// TIA Portal project "linia_do_napojow_V18" (V18)

(* hardware
DEVICE "S71500/ET200MP station_1"  S7-1500 station
   slot 0: "Rail_0"  Rack  6ES7 590-1***0-0AA0
   slot 1: "PLC_1"  CPU 1516-3 PN/DP  6ES7 516-3AN02-0AB0  V2.8
      slot 3: "CPU display_1"  6ES7591-1BA00-0AA0
      slot 32768: "PROFINET interface_1"  X1
         slot 32769: "Port_1"  X1 P1
         slot 32770: "Port_2"  X1 P2
      slot 33024: "PROFINET interface_2"  X2
         slot 33025: "Port_1"  X2 P1
      slot 33280: "DP interface_1"  X3
      slot 34817: "Virtual CP interface port_1"  Virtual CP interface port  Virtual CP interface port
   slot 2: "DI 32x24VDC HF_1"  DI 32x24VDC HF  6ES7 521-1BL00-0AB0  V2.2
   slot 3: "DQ 32x24VDC/0.5A HF_1"  DQ 32x24VDC/0.5A HF  6ES7 522-1BL01-0AB0  V1.1
   slot 4: "AI 8xU/I/RTD/TC ST_1"  AI 8xU/I/RTD/TC ST  6ES7 531-7KF00-0AB0  V2.2
   slot 5: "AQ 4xU/I ST_1"  AQ 4xU/I ST  6ES7 532-5HD00-0AB0  V2.2
DEVICE "HMI_1"  KTP900 Basic PN
   slot 0: "HMI_1"  KTP900 Basic PN  6AV2 123-2JB03-0AX0  16.0.0.0
   slot 1: "HMI_RT_1"  KTP900 Basic PN  6AV2 123-2JB03-0AX0  16.0.0.0
   slot 5: "HMI_1.IE_CP_1"  PROFINET Interface  16.0.0.0
      slot 1: "PROFINET Interface_1"  PROFINET Interface
         slot 1: "Port_1"  Port
*)

// ===== PLC "PLC_1"  CPU 1516-3 PN/DP =====

VAR_GLOBAL   // PLC tag table "Default tag table"
   "System_Byte" AT %MB1 : Byte;
   "FirstScan" AT %M1.0 : Bool;
   "DiagStatusUpdate" AT %M1.1 : Bool;
   "AlwaysTRUE" AT %M1.2 : Bool;
   "AlwaysFALSE" AT %M1.3 : Bool;
   "Clock_Byte" AT %MB0 : Byte;
   "Clock_10Hz" AT %M0.0 : Bool;
   "Clock_5Hz" AT %M0.1 : Bool;
   "Clock_2.5Hz" AT %M0.2 : Bool;
   "Clock_2Hz" AT %M0.3 : Bool;
   "Clock_1.25Hz" AT %M0.4 : Bool;
   "Clock_1Hz" AT %M0.5 : Bool;
   "Clock_0.625Hz" AT %M0.6 : Bool;
   "Clock_0.5Hz" AT %M0.7 : Bool;
   "rozlaczenie_tasmy" AT %M100.2 : Bool;
   "reset_licznika" AT %M100.3 : Bool;
   "zatrzymanie_tasmy" AT %M101.2 : Bool;
   "ilosc_butelek" AT %MW10 : Int;
   "reset_licznika_zak" AT %M101.3 : Bool;
   "ilosc_butelek_zak" AT %MW16 : Int;
   "Wylacznik_bezpieczenstwa" AT %M205.0 : Bool;
   "Wlacznik/Wylacznik_glowny" AT %M206.0 : Bool;
   "start_przenosik" AT %M204.0 : Bool;
   "stop_przenosnik" AT %M204.1 : Bool;
   "przenosnik_tasmowy" AT %Q1.4 : Bool;
   "wylacznik_przenosnika_tasmowego" AT %I1.4 : Bool;
   "wylacznik_nalewarki" AT %I1.5 : Bool;
   "wylacznik_zakrecarki" AT %I1.6 : Bool;
   "wylacznik_etykieciarki" AT %I1.7 : Bool;
   "wylacznik_pakowanie" AT %I2.0 : Bool;
   "samopod_start_zak" AT %M102.3 : Bool;
   "samopod_start_nal" AT %M100.4 : Bool;
   "Wlacznik_500ml" AT %M207.0 : Bool;
   "silownik" AT %Q1.5 : Bool;
   "sygnalizator_dzwiekowy" AT %Q2.2 : Bool;
   "robot" AT %Q2.3 : Bool;
   "lampa_przenosnik" AT %Q2.4 : Bool;
   "licznik_etykiet" AT %MW50 : Int;
   "cz_poj_ety" AT %M210.0 : Bool;
   "reset_licznika_etyk" AT %M211.0 : Bool;
   "pamiec_smakow" AT %M100.5 : Bool;
   "smak_zatrzymaj" AT %M212.2 : Bool;
   "czas_nalewarka" AT %MD300 : Time;
   "czas_pakowanie" AT %MD304 : Time;
   "czas_zakrecarka" AT %MD308 : Time;
   "cz_butelek_pakowanie" AT %M230.0 : Bool;
   "Tag_1" AT %MW400 : Word;
   "licznik_przenosnik" AT %MW30 : Int;
   "res_licz_przen" AT %M350.0 : Bool;
   "Tag_4" AT %MD32 : Time;
   "Tag_5" AT %M500.0 : Bool;
   "res_licz_nalew" AT %M350.1 : Bool;
   "licznik_nalewarak" AT %MW34 : Int;
   "Tag_2" AT %M350.2 : Bool;
   "Tag_3" AT %MW38 : Word;
   "czas_move" AT %MD312 : DWord;
   "czas_w_int" AT %MD316 : UDInt;
   "Tag_6" AT %M320.0 : Bool;
   "Tag_7" AT %MD321 : Time;
   "Tag_8" AT %MD325 : Time;
   "Tag_9" AT %MD329 : DInt;
   "Tag_10" AT %I90.0 : Bool;
END_VAR

VAR_GLOBAL   // PLC tag table "Nalewarka"
   "start_nalewarka" AT %M100.0 : Bool;
   "stop_nalewarka" AT %M100.1 : Bool;
   "cz_pojemnosciowy" AT %M200.0 : Bool;
   "dozy" AT %Q0.1 : Bool;
   "tasma" AT %Q0.0 : Bool;
   "lampa" AT %Q0.2 : Bool;
   "wl_pomarancza" AT %M212.0 : Bool;
   "pomarancza" AT %Q2.5 : Bool;
   "wl_truskawka" AT %M212.1 : Bool;
   "truskawka" AT %Q2.6 : Bool;
   "cz_poz_napoju" AT %M213.0 : Bool;
END_VAR

VAR_GLOBAL   // PLC tag table "Zakrecarka"
   "start_zakrecarka" AT %M101.0 : Bool;
   "stop_zakrecarka" AT %M101.1 : Bool;
   "cz_pojemnosciowy_zak" AT %M201.0 : Bool;
   "tasma_zakrecarka" AT %Q0.4 : Bool;
   "zakretka" AT %Q0.3 : Bool;
   "lampa_sygnalizacyjna" AT %Q0.5 : Bool;
END_VAR

VAR_GLOBAL   // PLC tag table "Etykieciarka"
   "start_etykieciarka" AT %M102.0 : Bool;
   "stop_etykieciarka" AT %M102.1 : Bool;
   "cz_swiatlowodowy" AT %M202.0 : Bool;
   "etykieta" AT %Q0.6 : Bool;
   "tasma_etykieciarka" AT %Q0.7 : Bool;
   "lampa_sygnalizacyjna_etyk" AT %Q1.0 : Bool;
END_VAR

VAR_GLOBAL   // PLC tag table "Pakowanie"
   "start_pakowaie" AT %M103.0 : Bool;
   "stop_pakowanie" AT %M103.1 : Bool;
   "cz_pojemnosciowy_pak" AT %M203.0 : Bool;
   "tasma_pakowanie" AT %Q1.2 : Bool;
   "lampa_sygnalizacyjna_pak" AT %Q1.1 : Bool;
   "cz_do_robota" AT %Q1.3 : Bool;
END_VAR

DATA_BLOCK "Nalewarka_DB"   // DB3
{ S7_Optimized_Access := 'TRUE' }
VERSION : 0.1
// stored: InstanceOfName Nalewarka
"Nalewarka"
BEGIN
END_DATA_BLOCK

DATA_BLOCK "Zakrecarka_DB"   // DB6
{ S7_Optimized_Access := 'TRUE' }
VERSION : 0.1
// stored: InstanceOfName Zakrecarka
"Zakrecarka"
BEGIN
END_DATA_BLOCK

DATA_BLOCK "Etykieciarka_DB"   // DB7
{ S7_Optimized_Access := 'TRUE' }
VERSION : 0.1
// stored: InstanceOfName Etykieciarka
"Etykieciarka"
BEGIN
END_DATA_BLOCK

DATA_BLOCK "Pakowanie_DB"   // DB9
{ S7_Optimized_Access := 'TRUE' }
VERSION : 0.1
// stored: InstanceOfName Pakowanie
"Pakowanie"
BEGIN
END_DATA_BLOCK

DATA_BLOCK "Przenosnik tasmowy_DB"   // DB12
{ S7_Optimized_Access := 'TRUE' }
VERSION : 0.1
// stored: InstanceOfName Przenosnik tasmowy
"Przenosnik tasmowy"
BEGIN
END_DATA_BLOCK

// folder: System blocks/Program resources

DATA_BLOCK "IEC_Counter_0_DB"   // DB1
{ S7_Optimized_Access := 'TRUE' }
AUTHOR : Simatic
FAMILY : IEC
NAME : CNTR
VERSION : 1.0
// stored: InstanceOfName IEC_COUNTER
"IEC_COUNTER"
BEGIN
END_DATA_BLOCK

DATA_BLOCK "IEC_Timer_0_DB"   // DB2
{ S7_Optimized_Access := 'TRUE' }
AUTHOR : Simatic
FAMILY : IEC
NAME : IEC_TMR
VERSION : 1.0
// stored: InstanceOfName IEC_TIMER
"IEC_TIMER"
BEGIN
END_DATA_BLOCK

DATA_BLOCK "IEC_Counter_0_DB_1"   // DB4
{ S7_Optimized_Access := 'TRUE' }
AUTHOR : Simatic
FAMILY : IEC
NAME : CNTR
VERSION : 1.0
// stored: InstanceOfName IEC_COUNTER
"IEC_COUNTER"
BEGIN
END_DATA_BLOCK

DATA_BLOCK "IEC_Timer_0_DB_1"   // DB5
{ S7_Optimized_Access := 'TRUE' }
AUTHOR : Simatic
FAMILY : IEC
NAME : IEC_TMR
VERSION : 1.0
// stored: InstanceOfName IEC_TIMER
"IEC_TIMER"
BEGIN
END_DATA_BLOCK

DATA_BLOCK "IEC_Counter_0_DB_2"   // DB8
{ S7_Optimized_Access := 'TRUE' }
AUTHOR : Simatic
FAMILY : IEC
NAME : CNTR
VERSION : 1.0
// stored: InstanceOfName IEC_COUNTER
"IEC_COUNTER"
BEGIN
END_DATA_BLOCK

DATA_BLOCK "IEC_Timer_0_DB_2"   // DB10
{ S7_Optimized_Access := 'TRUE' }
AUTHOR : Simatic
FAMILY : IEC
NAME : IEC_TMR
VERSION : 1.0
// stored: InstanceOfName IEC_TIMER
"IEC_TIMER"
BEGIN
END_DATA_BLOCK

// folder: (top level)

FUNCTION_BLOCK "Nalewarka"   // FB1, LAD
{ S7_Optimized_Access := 'TRUE' }
VERSION : 0.1
   VAR
      czas_nalewarka : Time;
   END_VAR
   VAR_TEMP   // added for the SCL form of the ladder/FBD networks
      _w1 : Bool;
   END_VAR
BEGIN

REGION Network 1
   // Start przenośnika taśmowego i zapalenie się lampy sygnalizacyjnej.
   // Wyłącznik nalewarki znajduje się fizycznie na linii produkcyjnej, w jego skład wchodzi również system ryglowania. Stop natomiast w panelu HMI.
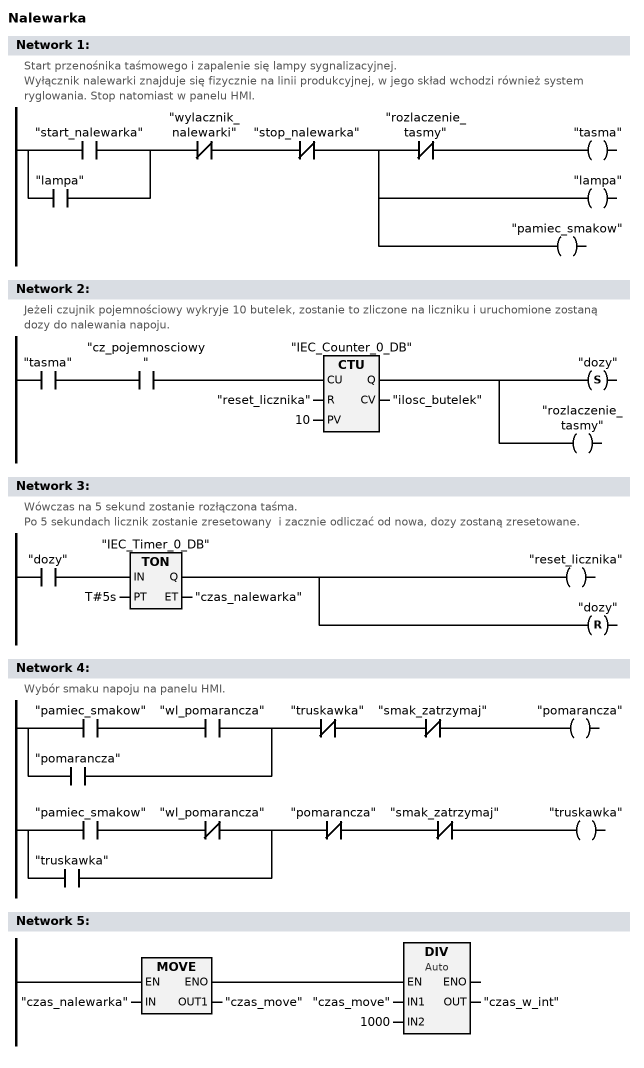
   RUNG wire#powerrail
      Contact( "start_nalewarka" )
      wire#w1
      I_Contact( "wylacznik_nalewarki" )
      I_Contact( "stop_nalewarka" )
      wire#w2
      I_Contact( "rozlaczenie_tasmy" )
      Coil( "tasma" )
   END_RUNG
   RUNG wire#powerrail
      Contact( "lampa" )
   END_RUNG wire#w1
   RUNG wire#w2
      Coil( "lampa" )
   END_RUNG
   RUNG wire#w2
      Coil( "pamiec_smakow" )
   END_RUNG
   // the same network as SCL:
   #_w1 := ("start_nalewarka" OR "lampa") AND NOT "wylacznik_nalewarki" AND NOT "stop_nalewarka";
   "tasma" := #_w1 AND NOT "rozlaczenie_tasmy";
   "lampa" := #_w1;
   "pamiec_smakow" := #_w1;
END_REGION

REGION Network 2
   // Jeżeli czujnik pojemnościowy wykryje 10 butelek, zostanie to zliczone na liczniku i uruchomione zostaną dozy do nalewania napoju.
   "IEC_Counter_0_DB".CTU(CU := "tasma" AND "cz_pojemnosciowy",
                          R := "reset_licznika",
                          PV := 10,
                          CV => "ilosc_butelek");
   IF "IEC_Counter_0_DB".Q THEN "dozy" := TRUE; END_IF;
   "rozlaczenie_tasmy" := "IEC_Counter_0_DB".Q;
END_REGION

REGION Network 3
   // Wówczas na 5 sekund zostanie rozłączona taśma.
   // Po 5 sekundach licznik zostanie zresetowany  i zacznie odliczać od nowa, dozy zostaną zresetowane.
   "IEC_Timer_0_DB".TON(IN := "dozy", PT := T#5s, ET => "czas_nalewarka");
   "reset_licznika" := "IEC_Timer_0_DB".Q;
   IF "IEC_Timer_0_DB".Q THEN "dozy" := FALSE; END_IF;
END_REGION

REGION Network 4
   // Wybór smaku napoju na panelu HMI.
   RUNG wire#powerrail
      Contact( "pamiec_smakow" )
      Contact( "wl_pomarancza" )
      wire#w1
      I_Contact( "truskawka" )
      I_Contact( "smak_zatrzymaj" )
      Coil( "pomarancza" )
   END_RUNG
   RUNG wire#powerrail
      Contact( "pomarancza" )
   END_RUNG wire#w1
   RUNG wire#powerrail
      Contact( "pamiec_smakow" )
      I_Contact( "wl_pomarancza" )
      wire#w2
      I_Contact( "pomarancza" )
      I_Contact( "smak_zatrzymaj" )
      Coil( "truskawka" )
   END_RUNG
   RUNG wire#powerrail
      Contact( "truskawka" )
   END_RUNG wire#w2
   // the same network as SCL:
   "pomarancza" := (("pamiec_smakow" AND "wl_pomarancza") OR "pomarancza") AND NOT "truskawka" AND NOT "smak_zatrzymaj";
   "truskawka" := (("pamiec_smakow" AND NOT "wl_pomarancza") OR "truskawka") AND NOT "pomarancza" AND NOT "smak_zatrzymaj";
END_REGION

REGION Network 5
   RUNG wire#powerrail
      Move(in := "czas_nalewarka", out1 => "czas_move")
      Div(in1 := "czas_move", in2 := 1000, out => "czas_w_int")
   END_RUNG
   // the same network as SCL:
   "czas_move" := "czas_nalewarka";
   "czas_w_int" := "czas_move" / 1000;
END_REGION
END_FUNCTION_BLOCK

FUNCTION_BLOCK "Zakrecarka"   // FB2, LAD
{ S7_Optimized_Access := 'TRUE' }
VERSION : 0.1
   VAR_TEMP   // added for the SCL form of the ladder/FBD networks
      _w1 : Bool;
   END_VAR
BEGIN

REGION Network 1
   // Start przenośnika taśmowego i zapalenie się lampy sygnalizacyjnej.
   // Wyłącznik zakręcarki znajduje się fizycznie na linii produkcyjnej, w jego skład wchodzi również system ryglowania. Stop natomiast w panelu HMI.
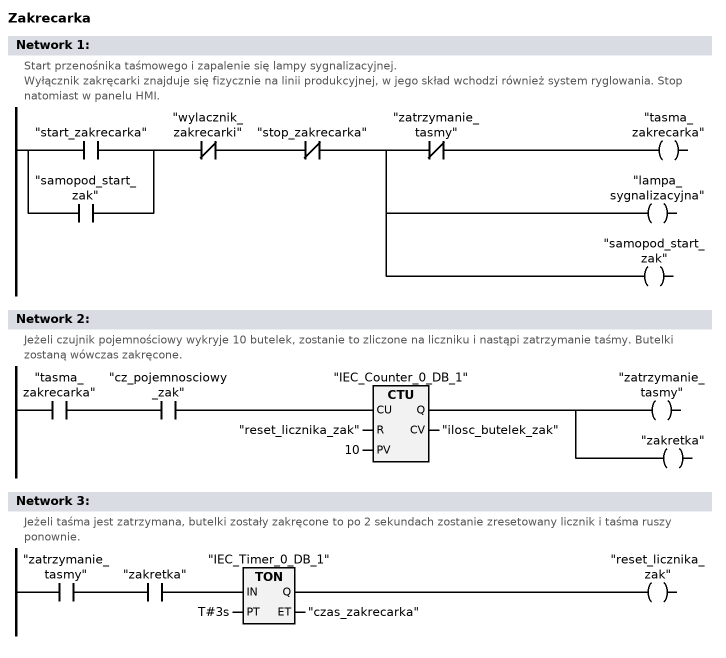
   RUNG wire#powerrail
      Contact( "start_zakrecarka" )
      wire#w1
      I_Contact( "wylacznik_zakrecarki" )
      I_Contact( "stop_zakrecarka" )
      wire#w2
      I_Contact( "zatrzymanie_tasmy" )
      Coil( "tasma_zakrecarka" )
   END_RUNG
   RUNG wire#powerrail
      Contact( "samopod_start_zak" )
   END_RUNG wire#w1
   RUNG wire#w2
      Coil( "lampa_sygnalizacyjna" )
   END_RUNG
   RUNG wire#w2
      Coil( "samopod_start_zak" )
   END_RUNG
   // the same network as SCL:
   #_w1 := ("start_zakrecarka" OR "samopod_start_zak") AND NOT "wylacznik_zakrecarki" AND NOT "stop_zakrecarka";
   "tasma_zakrecarka" := #_w1 AND NOT "zatrzymanie_tasmy";
   "lampa_sygnalizacyjna" := #_w1;
   "samopod_start_zak" := #_w1;
END_REGION

REGION Network 2
   // Jeżeli czujnik pojemnościowy wykryje 10 butelek, zostanie to zliczone na liczniku i nastąpi zatrzymanie taśmy. Butelki zostaną wówczas zakręcone.
   "IEC_Counter_0_DB_1".CTU(CU := "tasma_zakrecarka" AND "cz_pojemnosciowy_zak",
                           R := "reset_licznika_zak",
                           PV := 10,
                           CV => "ilosc_butelek_zak");
   "zatrzymanie_tasmy" := "IEC_Counter_0_DB_1".Q;
   "zakretka" := "IEC_Counter_0_DB_1".Q;
END_REGION

REGION Network 3
   // Jeżeli taśma jest zatrzymana, butelki zostały zakręcone to po 2 sekundach zostanie zresetowany licznik i taśma ruszy ponownie.
   "IEC_Timer_0_DB_1".TON(IN := "zatrzymanie_tasmy" AND "zakretka", PT := T#3s, ET => "czas_zakrecarka");
   "reset_licznika_zak" := "IEC_Timer_0_DB_1".Q;
END_REGION
END_FUNCTION_BLOCK

FUNCTION_BLOCK "Etykieciarka"   // FB3, LAD
{ S7_Optimized_Access := 'TRUE' }
VERSION : 0.1
BEGIN

REGION Network 1
   // Start przenośnika taśmowego i zapalenie się lampy sygnalizacyjnej.
   // Wyłącznik etykieciarki znajduje się fizycznie na linii produkcyjnej. Stop natomiast w panelu HMI.
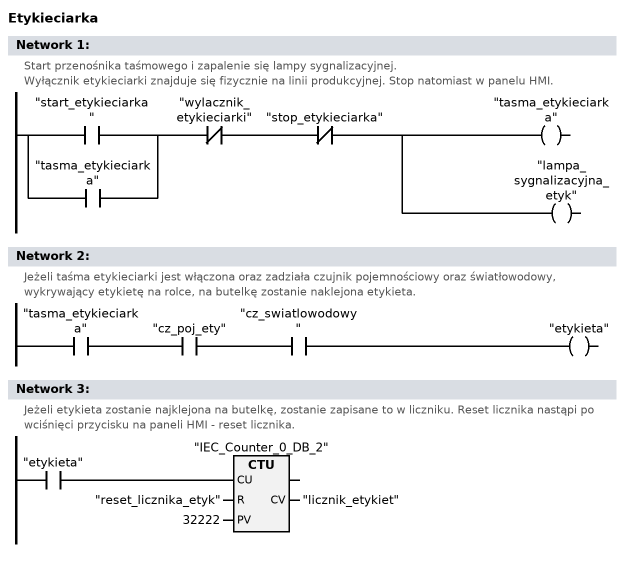
   RUNG wire#powerrail
      Contact( "start_etykieciarka" )
      wire#w1
      I_Contact( "wylacznik_etykieciarki" )
      I_Contact( "stop_etykieciarka" )
      wire#w2
      Coil( "tasma_etykieciarka" )
   END_RUNG
   RUNG wire#powerrail
      Contact( "tasma_etykieciarka" )
   END_RUNG wire#w1
   RUNG wire#w2
      Coil( "lampa_sygnalizacyjna_etyk" )
   END_RUNG
   // the same network as SCL:
   "tasma_etykieciarka" := ("start_etykieciarka" OR "tasma_etykieciarka") AND NOT "wylacznik_etykieciarki" AND NOT "stop_etykieciarka";
   "lampa_sygnalizacyjna_etyk" := "tasma_etykieciarka";
END_REGION

REGION Network 2
   // Jeżeli taśma etykieciarki jest włączona oraz zadziała czujnik pojemnościowy oraz światłowodowy, wykrywający etykietę na rolce, na butelkę zostanie naklejona etykieta.
   RUNG wire#powerrail
      Contact( "tasma_etykieciarka" )
      Contact( "cz_poj_ety" )
      Contact( "cz_swiatlowodowy" )
      Coil( "etykieta" )
   END_RUNG
   // the same network as SCL:
   "etykieta" := "tasma_etykieciarka" AND "cz_poj_ety" AND "cz_swiatlowodowy";
END_REGION

REGION Network 3
   // Jeżeli etykieta zostanie najklejona na butelkę, zostanie zapisane to w liczniku. Reset licznika nastąpi po wciśnięci przycisku na paneli HMI - reset licznika.
   "IEC_Counter_0_DB_2".CTU(CU := "etykieta", R := "reset_licznika_etyk", PV := 32222, CV => "licznik_etykiet");
END_REGION
END_FUNCTION_BLOCK

FUNCTION_BLOCK "Pakowanie"   // FB4, LAD
{ S7_Optimized_Access := 'TRUE' }
VERSION : 0.1
BEGIN

REGION Network 1
   // Start przenośnika taśmowego i zapalenie się lampy sygnalizacyjnej.
   // Wyłącznik pakowania znajduje się fizycznie na linii produkcyjnej, w jego skład wchodzi również kurtyna świetlna. Stop natomiast w panelu HMI.
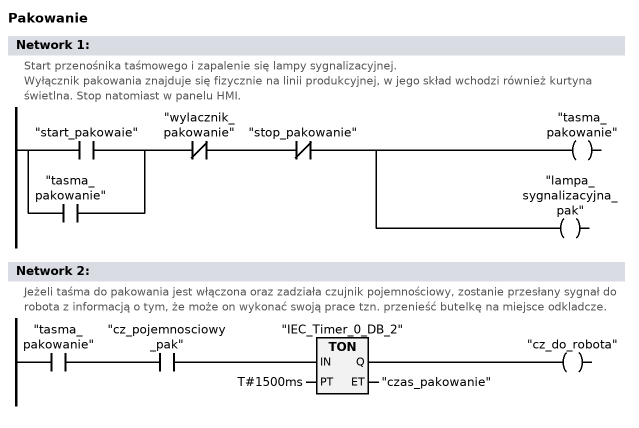
   RUNG wire#powerrail
      Contact( "start_pakowaie" )
      wire#w1
      I_Contact( "wylacznik_pakowanie" )
      I_Contact( "stop_pakowanie" )
      wire#w2
      Coil( "tasma_pakowanie" )
   END_RUNG
   RUNG wire#powerrail
      Contact( "tasma_pakowanie" )
   END_RUNG wire#w1
   RUNG wire#w2
      Coil( "lampa_sygnalizacyjna_pak" )
   END_RUNG
   // the same network as SCL:
   "tasma_pakowanie" := ("start_pakowaie" OR "tasma_pakowanie") AND NOT "wylacznik_pakowanie" AND NOT "stop_pakowanie";
   "lampa_sygnalizacyjna_pak" := "tasma_pakowanie";
END_REGION

REGION Network 2
   // Jeżeli taśma do pakowania jest włączona oraz zadziała czujnik pojemnościowy, zostanie przesłany sygnał do robota z informacją o tym, że może on wykonać swoją prace tzn. przenieść butelkę na miejsce odkladcze.
   "IEC_Timer_0_DB_2".TON(IN := "tasma_pakowanie" AND "cz_pojemnosciowy_pak",
                          PT := T#1500ms,
                          ET => "czas_pakowanie");
   "cz_do_robota" := "IEC_Timer_0_DB_2".Q;
END_REGION
END_FUNCTION_BLOCK

FUNCTION_BLOCK "Przenosnik tasmowy"   // FB5, LAD
{ S7_Optimized_Access := 'TRUE' }
VERSION : 0.1
   VAR_TEMP
      mem0 : Time;
   END_VAR
BEGIN

REGION Network 1
   // Start przenośnika taśmowego.
   // Wyłącznik przenośnika znajduje się fizycznie na linii produkcyjnej. Stop natomiast w panelu HMI.
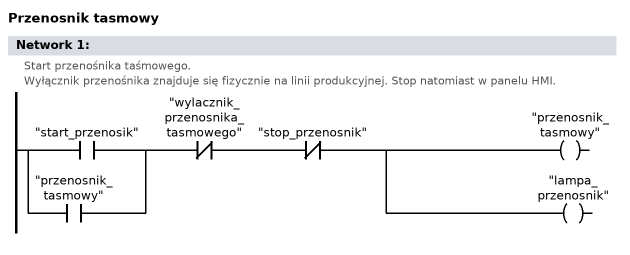
   RUNG wire#powerrail
      Contact( "start_przenosik" )
      wire#w1
      I_Contact( "wylacznik_przenosnika_tasmowego" )
      I_Contact( "stop_przenosnik" )
      wire#w2
      Coil( "przenosnik_tasmowy" )
   END_RUNG
   RUNG wire#powerrail
      Contact( "przenosnik_tasmowy" )
   END_RUNG wire#w1
   RUNG wire#w2
      Coil( "lampa_przenosnik" )
   END_RUNG
   // the same network as SCL:
   "przenosnik_tasmowy" := ("start_przenosik" OR "przenosnik_tasmowy") AND NOT "wylacznik_przenosnika_tasmowego" AND NOT "stop_przenosnik";
   "lampa_przenosnik" := "przenosnik_tasmowy";
END_REGION
END_FUNCTION_BLOCK

ORGANIZATION_BLOCK "Main"   // OB1, LAD, ProgramCycle
TITLE = "Main Program Sweep (Cycle)"
{ S7_Optimized_Access := 'TRUE' }
VERSION : 0.1
   VAR_INPUT
      Initial_Call : Bool;   // Initial call of this OB
      Remanence : Bool;   // =True, if remanent data are available
   END_VAR
   VAR_TEMP   // added for the SCL form of the ladder/FBD networks
      _w1 : Bool;
      _w2 : Bool;
      _w3 : Bool;
      _w4 : Bool;
      _w5 : Bool;
   END_VAR
BEGIN

REGION Network 1
   // Linię produkcyjną uruchamiamy poprzez włącznik główny oraz dodatkowo każdy etap produkcji na panelu HMI.
   // Wyłącznik bezpieczeństwa znajduje się w kilku miejscach na linii produkcyjnej.
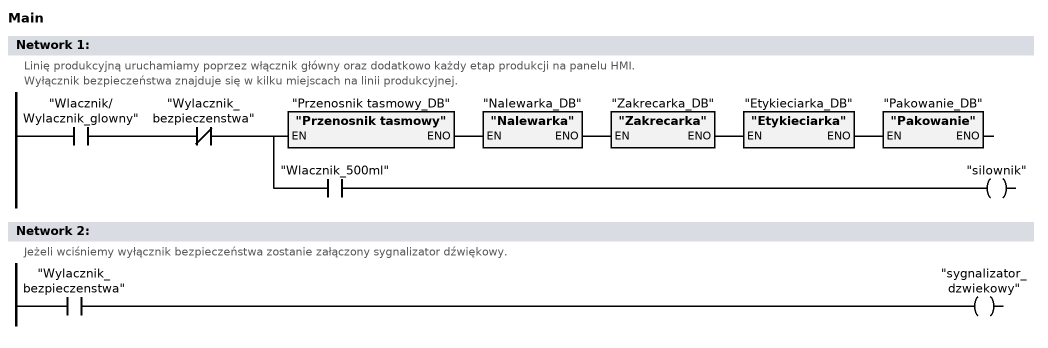
   RUNG wire#powerrail
      Contact( "Wlacznik/Wylacznik_glowny" )
      I_Contact( "Wylacznik_bezpieczenstwa" )
      wire#w1
      "Przenosnik tasmowy_DB"()
      "Nalewarka_DB"()
      "Zakrecarka_DB"()
      "Etykieciarka_DB"()
      "Pakowanie_DB"()
   END_RUNG
   RUNG wire#w1
      Contact( "Wlacznik_500ml" )
      Coil( "silownik" )
   END_RUNG
   // the same network as SCL:
   #_w1 := "Wlacznik/Wylacznik_glowny" AND NOT "Wylacznik_bezpieczenstwa";
   "Przenosnik tasmowy_DB"(EN := #_w1, ENO => #_w2);   // "Przenosnik tasmowy"
   "Nalewarka_DB"(EN := #_w2, ENO => #_w3);   // "Nalewarka"
   "Zakrecarka_DB"(EN := #_w3, ENO => #_w4);   // "Zakrecarka"
   "Etykieciarka_DB"(EN := #_w4, ENO => #_w5);   // "Etykieciarka"
   IF #_w5 THEN
       "Pakowanie_DB"();   // "Pakowanie"
   END_IF;
   "silownik" := #_w1 AND "Wlacznik_500ml";
END_REGION

REGION Network 2
   // Jeżeli wciśniemy wyłącznik bezpieczeństwa zostanie załączony sygnalizator dźwiękowy.
   RUNG wire#powerrail
      Contact( "Wylacznik_bezpieczenstwa" )
      Coil( "sygnalizator_dzwiekowy" )
   END_RUNG
   // the same network as SCL:
   "sygnalizator_dzwiekowy" := "Wylacznik_bezpieczenstwa";
END_REGION
END_ORGANIZATION_BLOCK

(* ===== HMI "HMI_RT_1" =====
system functions are stored by id; their names below are inferred from use
connection "HMI_Connection_1": ETHERNET, SMART_S7_1500_OMS

HMI tags "Default tag table"
   "Wlacznik_glowny" : Bool = PLC "Wlacznik/Wylacznik_glowny" AT %M206.0, 1 s
   "start_przenosik" : Bool = PLC start_przenosik AT %M204.0, 1 s
   "stop_przenosnik" : Bool = PLC stop_przenosnik AT %M204.1, 1 s
   "przenosnik_tasmowy" : Bool = PLC przenosnik_tasmowy AT %Q1.4, 1 s
      on ChangeValue: function_b9b71300("MOVE(1)", 1)
   "start_nalewarka" : Bool = PLC start_nalewarka AT %M100.0, 1 s
   "stop_nalewarka" : Bool = PLC stop_nalewarka AT %M100.1, 1 s
   "start_zakrecarka" : Bool = PLC start_zakrecarka AT %M101.0, 1 s
   "stop_zakrecarka" : Bool = PLC stop_zakrecarka AT %M101.1, 1 s
   "start_etykieciarka" : Bool = PLC start_etykieciarka AT %M102.0, 1 s
   "stop_etykieciarka" : Bool = PLC stop_etykieciarka AT %M102.1, 1 s
   "start_pakowaie" : Bool = PLC start_pakowaie AT %M103.0, 1 s
   "stop_pakowanie" : Bool = PLC stop_pakowanie AT %M103.1, 1 s
   "silownik" : Bool = PLC silownik AT %Q1.5, 1 s
   "Wlacznik_500ml" : Bool = PLC Wlacznik_500ml AT %M207.0, 1 s
   "lampa" : Bool = PLC lampa AT %Q0.2, 1 s
   "lampa_sygnalizacyjna" : Bool = PLC lampa_sygnalizacyjna AT %Q0.5, 1 s
   "lampa_sygnalizacyjna_etyk" : Bool = PLC lampa_sygnalizacyjna_etyk AT %Q1.0, 1 s
   "lampa_sygnalizacyjna_pak" : Bool = PLC lampa_sygnalizacyjna_pak AT %Q1.1, 1 s
   "cz_do_robota" : Bool = PLC cz_do_robota AT %Q1.3, 1 s
   "tasma_pakowanie" : Bool = PLC tasma_pakowanie AT %Q1.2, 1 s
      on ChangeValue: function_b9b71300("move_pako", 1)
   "cz_pojemnosciowy" : Bool = PLC cz_pojemnosciowy AT %M200.0, 1 s
   "dozy" : Bool = PLC dozy AT %Q0.1, 1 s
   "tasma" : Bool = PLC tasma AT %Q0.0, 1 s
      on ChangeValue: function_b9b71300("MOVE_nal", 1)
   "ilosc_butelek" : Int = PLC ilosc_butelek AT %MW10, 1 s
   "cz_pojemnosciowy_pak" : Bool = PLC cz_pojemnosciowy_pak AT %M203.0, 1 s
   "lampa_przenosnik" : Bool = PLC lampa_przenosnik AT %Q2.4, 1 s
   "licznik_etykiet" : Int = PLC licznik_etykiet AT %MW50, 1 s
   "tasma_etykieciarka" : Bool = PLC tasma_etykieciarka AT %Q0.7, 1 s
      on ChangeValue: function_b9b71300("move_etyk", 1)
   "cz_poj_ety" : Bool = PLC cz_poj_ety AT %M210.0, 1 s
   "cz_swiatlowodowy" : Bool = PLC cz_swiatlowodowy AT %M202.0, 1 s
   "etykieta" : Bool = PLC etykieta AT %Q0.6, 1 s
   "reset_licznika_etyk" : Bool = PLC reset_licznika_etyk AT %M211.0, 1 s
   "ilosc_butelek_zak" : Int = PLC ilosc_butelek_zak AT %MW16, 1 s
   "tasma_zakrecarka" : Bool = PLC tasma_zakrecarka AT %Q0.4, 1 s
      on ChangeValue: function_b9b71300("move_zak", 1)
   "cz_pojemnosciowy_zak" : Bool = PLC cz_pojemnosciowy_zak AT %M201.0, 1 s
   "zakretka" : Bool = PLC zakretka AT %Q0.3, 1 s
   "wl_pomarancza" : Bool = PLC wl_pomarancza AT %M212.0, 1 s
   "sygnalizator_dzwiekowy" : Bool = PLC sygnalizator_dzwiekowy AT %Q2.2, 1 s
   "smak_zatrzymaj" : Bool = PLC smak_zatrzymaj AT %M212.2, 1 s
   "pomarancza" : Bool = PLC pomarancza AT %Q2.5, 1 s
   "truskawka" : Bool = PLC truskawka AT %Q2.6, 1 s
   "czas_pakowanie" : Time = PLC czas_pakowanie AT %MD304, 1 s
   "czas_zakrecarka" : Time = PLC czas_zakrecarka AT %MD308, 1 s
   "czas_nalewarka" : Time = PLC czas_nalewarka AT %MD300, 1 s
   "move" : Int, internal
   "Clock_Byte" : Byte = PLC Clock_Byte AT %MB0, 1 s
   "Tag_1" : Word = PLC Tag_1 AT %MW400, 1 s
   "Tag_2" : Int = PLC licznik_przenosnik AT %MW30, 1 s
   "Tag_4" : Time = PLC Tag_4 AT %MD32, 1 s
   "licznik_nalewarak" : Int = PLC licznik_nalewarak AT %MW34, 1 s
   "MOVE(1)" : Int, internal
   "MOVE_nal" : Int, internal
   "rozlaczenie_tasmy" : Bool = PLC rozlaczenie_tasmy AT %M100.2, 1 s
   "Tag_6" : DWord = PLC czas_move AT %MD312, 1 s
   "Tag_7" : UDInt = PLC czas_w_int AT %MD316, 1 s
   "move_etyk" : Int, internal
   "Tag_6(1)" : Bool = PLC Tag_6 AT %M320.0, 1 s
   "Tag_7(1)" : Time = PLC Tag_7 AT %MD321, 1 s
   "Tag_9" : DInt = PLC Tag_9 AT %MD329, 1 s
   "move_zak" : Int, internal
   "move_nal(1)" : Int, internal
   "move_pako" : Int, internal

text list "Lista": 0 'Butelki szklane - 250ml'; 1 'Butelki szklane - 500ml'

text list "Smaki": 0 'truskawkowy'; 1 'pomarańczowy'

text list "Ilosc_butelek": 1 '10'; 2 '9'; 3 '8'; 4 '7'; 5 '6'; 6 '5'; 7 '4'; 8 '3'; 9 '2'; 10 '1'

Template "Template_1" 800x480
   Button "Exit" at 722,440 size 55x39; TextOff 'Exit'; PictureOff "ExitRuntime_KTP900_Basic_PN_TR"; PictureOn "ExitRuntime_KTP900_Basic_PN_TR"
      on Release: StopRuntime(0)
   Button "Template_Button" at 622,440 size 55x39; TextOff 'Text'
   Button "Template_Button_1" at 522,440 size 55x39; TextOff 'Text'
   Button "Template_Button_2" at 422,440 size 55x39; TextOff 'Text'
   Button "Template_Button_3" at 322,440 size 55x39; TextOff 'Text'
   Button "Template_Button_4" at 222,440 size 55x39; TextOff 'Text'
   Button "Alarms" at 122,440 size 55x39; TextOff 'Alarms'; PictureOff "AlarmDisplay_KTP900_Basic_PN_TR"; PictureOn "AlarmDisplay_KTP900_Basic_PN_TR"
      on Release: function_ef3f5d25("Alarm window_Unacknowledged", -1)
   Button "Start screen" at 22,440 size 55x39; TextOff 'Start screen'; PictureOff "NavigateHome_KTP900_Basic_PN_TR"; PictureOn "NavigateHome_KTP900_Basic_PN_TR"
      on Release: ActivateScreen("Wyswietlacz_glowny", 0)
   SymbolicIOField "Symbolic_IO_Field_Screen" at 73,7 size 620x26; TextOff '0'; TextOn '1'
   DateTimeField "HmiScreenItemData" at 695,20 size 105x20
   DateTimeField "HmiScreenItemData_1" at 695,0 size 105x20
   GraphicView "Logo" at 0,0 size 71x40; Picture "Logo of HMI_1"

screen "Wyswietlacz_glowny" 800x480, template "Template_1"
   Button "Button_1" at 22,48 size 355x82; TextOff 'Włącznik/Wyłącznik główny'
      on Click: InvertBit("Wlacznik_glowny")
      Appearance <- "Wlacznik_glowny"
   Button "Button_2" at 66,376 size 96x32; TextOff 'start'
      on Press: SetBit("start_nalewarka")
      on Release: ResetBit("start_nalewarka")
   Button "Button_3" at 66,270 size 96x32; TextOff 'start'; TextList "start"
      on Press: SetBit("start_przenosik")
      on Release: ResetBit("start_przenosik")
   Button "Button_4" at 254,270 size 96x32; TextOff 'stop'
      on Press: SetBit("stop_przenosnik")
      on Release: ResetBit("stop_przenosnik")
   TextField "Text field_1" at 128,220 size 153x29; Text 'Stół obrotowy'
   TextField "Text field_2" at 151,319 size 118x29; Text 'Nalewarka'
   TextField "Text field_3" at 548,78 size 123x29; Text 'Zakręcarka'
   TextField "Text field_4" at 537,190 size 134x29; Text 'Etykieciarka'
   TextField "Text field_5" at 548,322 size 120x29; Text 'Pakowanie'
   Button "Button_5" at 254,376 size 96x32; TextOff 'stop'
      on Press: SetBit("stop_nalewarka")
      on Release: ResetBit("stop_nalewarka")
   Button "Button_6" at 461,123 size 96x32; TextOff 'start'
      on Press: SetBit("start_zakrecarka")
      on Release: ResetBit("start_zakrecarka")
   Button "Button_7" at 651,123 size 96x32; TextOff 'stop'
      on Press: SetBit("stop_zakrecarka")
      on Release: ResetBit("stop_zakrecarka")
   Button "Button_8" at 461,244 size 96x32; TextOff 'start'
      on Press: SetBit("start_etykieciarka")
      on Release: ResetBit("start_etykieciarka")
   Button "Button_9" at 651,249 size 96x32; TextOff 'stop'
      on Press: SetBit("stop_etykieciarka")
      on Release: ResetBit("stop_etykieciarka")
   Button "Button_10" at 461,382 size 96x32; TextOff 'start'
      on Press: SetBit("start_pakowaie")
      on Release: ResetBit("start_pakowaie")
   Button "Button_11" at 651,382 size 96x32; TextOff 'stop'
      on Press: SetBit("stop_pakowanie")
      on Release: ResetBit("stop_pakowanie")
   Circle "Circle_2" at 182,372 size 48x48
      Appearance <- "lampa"
   Circle "Circle_3" at 582,116 size 48x48
      Appearance <- "lampa_sygnalizacyjna"
   Circle "Circle_4" at 582,235 size 48x48
      Appearance <- "lampa_sygnalizacyjna_etyk"
   Circle "Circle_5" at 582,374 size 48x48
      Appearance <- "lampa_sygnalizacyjna_pak"
   Circle "Circle_1" at 182,262 size 48x48
      Appearance <- "przenosnik_tasmowy"
   SymbolicIOField "Symbolic I/O field_2" at 22,146 size 232x53; TextOff '0'; TextOn '1'; TextList "Lista"
      ProcessValue <- "Wlacznik_500ml"
      on Change: SetBit("Wlacznik_500ml")
   GraphicView "Graphic view_2" at 399,43 size 88x59; Picture "Graphic_12"
   Button "Button_13" at 333,219 size 41x35; TextOff 'Przenosnik_tasmowy'; PictureOff "Graphic_8"
      on Click: ActivateScreen("Przenosnik_tasmowy", 0)
   Button "Button_17" at 691,314 size 41x35; TextOn 'Przenosnik_tasmowy'; TextOff 'Przenosnik_tasmowy'; PictureOff "Graphic_8"
      on Click: ActivateScreen("Pakowanie", 0)
   Button "Button_12" at 691,68 size 41x35; TextOn 'Przenosnik_tasmowy'; TextOff 'Przenosnik_tasmowy'; PictureOff "Graphic_8"
      on Click: ActivateScreen("Zakrecarka", 0)
   Button "Button_18" at 691,184 size 41x35; TextOn 'Przenosnik_tasmowy'; TextOff 'Przenosnik_tasmowy'; PictureOff "Graphic_8"
      on Click: ActivateScreen("Etykieciarka", 0)
   Button "Button_19" at 333,319 size 41x35; TextOn 'Przenosnik_tasmowy'; TextOff 'Przenosnik_tasmowy'; PictureOff "Graphic_8"
      on Click: ActivateScreen("Nalewarka", 0)
   Circle "Circle_6" at 472,37 size 18x18
      Appearance <- "sygnalizator_dzwiekowy"

screen "Przenosnik_tasmowy" 800x480
   on GenerateScreen: function_f9c01323("MOVE(1)", 1, 100, 0, 1)
   GraphicView "Graphic view_1" at 65,273 size 652x144; Picture "Graphic_11"
   TextField "Text field_1" at 148,34 size 153x29; Text 'Stół obrotowy'
   Circle "Circle_1" at 383,29 size 48x48
      Appearance <- "przenosnik_tasmowy"
   Button "Button_1" at 49,92 size 170x51; TextOff 'start'
      on Press: SetBit("start_przenosik")
      on Release: ResetBit("start_przenosik")
   Circle "Circle_2" at 61,273 size 48x48
      Appearance <- "lampa_przenosnik"
   Button "Button_2" at 237,92 size 170x51; TextOff 'stop'
      on Release: ResetBit("stop_przenosnik")
      on Press: SetBit("stop_przenosnik")
   Button "Button_3" at 22,17 size 57x51; TextOff 'Wyswietlacz_glowny'; PictureOff "Left_Arrow"
      on Click: ActivateScreen("Wyswietlacz_glowny", 0)
   GraphicView "Graphic view_2" at 199,236 size 43x95; Picture "Graphic_33"
      HorizontalMovement <- "MOVE(1)"
      Visibility <- "przenosnik_tasmowy"
   GraphicView "Graphic view_5" at 199,236 size 43x95; Picture "Graphic_33"
      Visibility <- "przenosnik_tasmowy"

screen "Nalewarka" 800x480
   on GenerateScreen: function_f9c01323("MOVE_nal", 1, 100, 0, 1)
   Button "Button_1" at 52,102 size 157x52; TextOff 'start'
      on Press: SetBit("start_nalewarka")
      on Release: ResetBit("start_nalewarka")
   Circle "Circle_1" at 340,32 size 48x48
      Appearance <- "lampa"
   TextField "Text field_1" at 154,36 size 149x37; Text 'Nalewarka'
   Circle "Circle_2" at 26,339 size 48x48
      Appearance <- "tasma"
   GraphicView "Graphic view_1" at 14,374 size 777x83; Picture "Graphic_11"
   Button "Button_2" at 239,102 size 157x52; TextOff 'stop'
      on Press: SetBit("stop_nalewarka")
      on Release: ResetBit("stop_nalewarka")
   GraphicView "Graphic view_2" at 439,181 size 78x138; Picture "Graphic_17"
   IOField "I/O field_1" at 563,57 size 126x34; FormatPattern 99
      ProcessValue <- "ilosc_butelek"
   Circle "Circle_3" at 458,227 size 33x33
      Appearance <- "dozy"
   GraphicView "Graphic view_4" at 239,356 size 36x35; Picture "Graphic_15"
   Circle "Circle_4" at 275,353 size 15x15
      Appearance <- "cz_pojemnosciowy"
   IOField "I/O field_2" at 563,97 size 126x34; FormatPattern 99999
      ProcessValue <- "czas_nalewarka"
   TextField "Text field_2" at 708,58 size 70x27; Text 'Licznik'
   TextField "Text field_3" at 708,96 size 59x27; Text 'Timer'
   Button "Button_3" at 27,20 size 56x49; TextOff 'Wyswietlacz_glowny'; PictureOff "Left_Arrow"
      on Click: ActivateScreen("Wyswietlacz_glowny", 0)
   SymbolicIOField "Symbolic I/O field_1" at 52,167 size 180x54; TextOn '1'; TextOff '0'; TextList "Smaki"
      on Change: SetBit("wl_pomarancza")
      ProcessValue <- "wl_pomarancza"
   GraphicView "Graphic view_6" at 403,57 size 65x95; Picture "Graphic_26"
   GraphicView "Graphic view_3" at 475,58 size 65x95; Picture "Graphic_26"
   Circle "Circle_5" at 428,74 size 34x34
      Appearance <- "pomarancza"
   Circle "Circle_6" at 497,72 size 34x34
      Appearance <- "truskawka"
   GraphicView "Graphic view_5" at 419,153 size 38x28; Picture "Graphic_28"
   GraphicView "Graphic view_9" at 453,151 size 38x33; Picture "Graphic_32"
   GraphicView "Graphic view_7" at 489,153 size 36x30; Picture "Graphic_30"
   Switch "Switch_1" at 52,235 size 113x40; CaptionText 'Switch'; TextOff 'stop'; TextOn 'start'
      ProcessValue <- "smak_zatrzymaj"
   TextField "Text field_4" at 177,244 size 157x25; Text 'Start/Stop smaku'
   GraphicView "Graphic view_8" at 106,319 size 43x95; Picture "Graphic_33"
      HorizontalMovement <- "MOVE_nal"
      Visibility <- "tasma"
   GraphicView "Graphic view_10" at 106,319 size 43x95; Picture "Graphic_33"
      Visibility <- "tasma"
   GraphicView "Graphic view_11" at 450,317 size 43x95; Picture "Graphic_33"
      Visibility <- "rozlaczenie_tasmy"
   Rectangle "Rectangle_1" at 453,391 size 37x15
      Visibility <- "Tag_7"
   Rectangle "Rectangle_2" at 453,376 size 37x15
      Visibility <- "Tag_7"
   Rectangle "Rectangle_3" at 453,362 size 37x15
      Visibility <- "Tag_7"
   Button "Button_4" at 625,228 size 96x32; TextOff 'czujnik'
      on Press: SetBit("cz_pojemnosciowy")
      on Release: ResetBit("cz_pojemnosciowy")
   SymbolicIOField "Symbolic I/O field_2" at 253,189 size 123x32; TextOff '0'; TextOn '1'; TextList "Ilosc_butelek"
   TextField "Text field_5" at 253,162 size 115x25; Text 'Ilość butelek'

screen "Zakrecarka" 800x480
   on GenerateScreen: function_f9c01323("move_zak", 1, 100, 0, 1)
   Button "Button_1" at 21,17 size 53x55; TextOff 'Wyswietlacz_glowny'; PictureOff "Left_Arrow"
      on Click: ActivateScreen("Wyswietlacz_glowny", 0)
   TextField "Text field_1" at 157,39 size 123x29; Text 'Zakręcarka'
   Circle "Circle_1" at 303,28 size 48x48
      Appearance <- "lampa_sygnalizacyjna"
   Button "Button_2" at 67,99 size 155x64; TextOff 'start'
      on Press: SetBit("start_zakrecarka")
      on Release: ResetBit("start_zakrecarka")
   GraphicView "Graphic view_1" at 9,315 size 768x113; Picture "Graphic_11"
   Button "Button_3" at 251,99 size 155x64; TextOff 'stop'
      on Press: SetBit("stop_zakrecarka")
      on Release: ResetBit("stop_zakrecarka")
   Circle "Circle_2" at 47,303 size 44x44
      Appearance <- "tasma_zakrecarka"
   GraphicView "Graphic view_4" at 324,302 size 36x35; Picture "Graphic_15"
   Circle "Circle_3" at 295,294 size 19x19
      Appearance <- "cz_pojemnosciowy_zak"
   TextField "Text field_2" at 659,68 size 70x27; Text 'Licznik'
   TextField "Text field_3" at 699,121 size 13x22; Text 'Text'
   IOField "I/O field_1" at 536,67 size 96x32; FormatPattern 99
      ProcessValue <- "ilosc_butelek_zak"
   IOField "I/O field_2" at 536,114 size 96x32; FormatPattern 99999
      ProcessValue <- "czas_zakrecarka"
   TextField "Text field_4" at 659,114 size 59x27; Text 'Timer'
   GraphicView "Graphic view_2" at 484,156 size 113x115; Picture "Graphic_24"
   Circle "Circle_4" at 525,187 size 29x29
      Appearance <- "zakretka"
   GraphicView "Graphic view_3" at 157,271 size 43x95; Picture "Graphic_33"
      HorizontalMovement <- "move_zak"
      Visibility <- "tasma_zakrecarka"
   Rectangle "Rectangle_4" at 160,315 size 37x44
      Visibility <- "tasma_zakrecarka"
      HorizontalMovement <- "move_zak"
   Button "Button_4" at 677,199 size 96x32; TextOff 'czujnik'
      on Press: SetBit("cz_pojemnosciowy_zak")
      on Release: ResetBit("cz_pojemnosciowy_zak")
   GraphicView "Graphic view_5" at 520,271 size 43x95; Picture "Graphic_33"
      Visibility <- "zakretka"
   Rectangle "Rectangle_1" at 523,313 size 37x44
      Visibility <- "zakretka"
   Rectangle "Rectangle_2" at 529,271 size 25x13
      Visibility <- "zakretka"

screen "Etykieciarka" 800x480
   on GenerateScreen: function_f9c01323("move_etyk", 1, 100, 0, 1)
   TextField "Text field_1" at 154,36 size 134x29; Text 'Etykieciarka'
   Circle "Circle_1" at 307,29 size 48x48
      Appearance <- "lampa_sygnalizacyjna_etyk"
   Button "Button_1" at 36,107 size 163x57; TextOff 'start'
      on Press: SetBit("start_etykieciarka")
      on Release: ResetBit("start_etykieciarka")
   GraphicView "Graphic view_1" at 0,337 size 787x115; Picture "Graphic_11"
   Circle "Circle_2" at 22,289 size 48x48
      Appearance <- "tasma_etykieciarka"
   Button "Button_2" at 472,93 size 152x43; TextOff 'Reset licznika'
      on Press: SetBit("reset_licznika_etyk")
      on Release: ResetBit("reset_licznika_etyk")
   IOField "I/O field_1" at 473,142 size 153x48; FormatPattern 999
      ProcessValue <- "licznik_etykiet"
   TextField "Text field_2" at 637,152 size 142x27; Text 'Licznik etykiet'
   Button "Button_3" at 215,109 size 163x57; TextOff 'start'
      on Release: ResetBit("stop_etykieciarka")
      on Press: SetBit("stop_etykieciarka")
   GraphicView "Graphic view_2" at 428,303 size 45x54; Picture "Graphic_19"
   GraphicView "Graphic view_4" at 431,321 size 36x35; Picture "Graphic_15"
   Circle "Circle_3" at 413,300 size 12x12
      Appearance <- "cz_poj_ety"
   Circle "Circle_4" at 415,329 size 13x13
      Appearance <- "cz_swiatlowodowy"
   GraphicView "Graphic view_3" at 473,302 size 67x57; Picture "Graphic_20"
   Circle "Circle_5" at 493,315 size 29x29
      Appearance <- "etykieta"
   Button "Button_4" at 22,19 size 61x53; TextOff 'Wyswietlacz_glowny'; PictureOff "Left_Arrow"
      on Click: ActivateScreen("Wyswietlacz_glowny", 0)
   Button "Button_5" at 611,213 size 96x32; TextOff 'Text'
      on Press: SetBit("cz_swiatlowodowy")
      on Release: ResetBit("cz_swiatlowodowy")
   GraphicView "Graphic view_5" at 206,292 size 43x95; Picture "Graphic_33"
      HorizontalMovement <- "move_etyk"
      Visibility <- "tasma_etykieciarka"
   Rectangle "Rectangle_1" at 208,335 size 39x46
      Visibility <- "tasma_etykieciarka"
      HorizontalMovement <- "move_etyk"
   Rectangle "Rectangle_2" at 215,289 size 26x16
      HorizontalMovement <- "move_etyk"
      Visibility <- "tasma_etykieciarka"
   GraphicView "Graphic view_6" at 486,292 size 43x95; Picture "Graphic_33"
      Visibility <- "etykieta"
   Rectangle "Rectangle_3" at 487,335 size 39x46
      Visibility <- "etykieta"
   Rectangle "Rectangle_4" at 494,289 size 26x16
      Visibility <- "etykieta"
   GraphicView "Graphic view_7" at 485,338 size 44x42; Picture "Graphic_40"
      Visibility <- "etykieta"

screen "Pakowanie" 800x480
   on GenerateScreen: function_f9c01323("move_pako", 1, 100, 0, 1)
   Button "Button_1" at 37,102 size 178x66; TextOff 'start'
      on Press: SetBit("start_pakowaie")
      on Release: ResetBit("start_pakowaie")
   Button "Button_2" at 231,103 size 178x65; TextOff 'stop'
      on Press: SetBit("stop_pakowanie")
      on Release: ResetBit("stop_pakowanie")
   GraphicView "Graphic view_1" at 37,327 size 404x115; Picture "Graphic_11"
   Circle "Circle_1" at 360,27 size 49x49
      Appearance <- "lampa_sygnalizacyjna_pak"
   Circle "Circle_2" at 409,214 size 48x48
      Appearance <- "cz_do_robota"
   Circle "Circle_3" at 17,281 size 48x48
      Appearance <- "tasma_pakowanie"
   TextField "Text field_1" at 159,34 size 152x37; Text 'Pakowanie'
   GraphicView "Graphic view_4" at 347,312 size 36x35; Picture "Graphic_15"
   Circle "Circle_4" at 383,293 size 24x24
      Appearance <- "cz_pojemnosciowy_pak"
   IOField "I/O field_1" at 503,56 size 112x47; FormatPattern 99999
      ProcessValue <- "czas_pakowanie"
   TextField "Text field_2" at 636,71 size 59x27; Text 'Timer'
   Button "Button_3" at 24,28 size 58x51; TextOff 'Wyswietlacz_glowny'; PictureOff "Left_Arrow"
      on Click: ActivateScreen("Wyswietlacz_glowny", 0)
   GraphicView "Graphic view_6" at 120,293 size 43x95; Picture "Graphic_33"
      HorizontalMovement <- "move_pako"
      Visibility <- "tasma_pakowanie"
   Rectangle "Rectangle_3" at 121,336 size 39x46
      HorizontalMovement <- "move_pako"
      Visibility <- "tasma_pakowanie"
   Rectangle "Rectangle_4" at 127,290 size 26x16
      HorizontalMovement <- "move_pako"
      Visibility <- "tasma_pakowanie"
   GraphicView "Graphic view_7" at 119,339 size 44x42; Picture "Graphic_40"
      HorizontalMovement <- "move_pako"
      Visibility <- "tasma_pakowanie"
   GraphicView "Graphic view_3" at 336,294 size 43x95; Picture "Graphic_33"
      Visibility <- "cz_pojemnosciowy_pak"
   Rectangle "Rectangle_1" at 337,337 size 39x46
      Visibility <- "cz_pojemnosciowy_pak"
   Rectangle "Rectangle_2" at 344,291 size 26x16
      Visibility <- "cz_pojemnosciowy_pak"
   GraphicView "Graphic view_5" at 335,340 size 44x42; Picture "Graphic_40"
      Visibility <- "cz_pojemnosciowy_pak"
   GraphicView "Graphic view_2" at 473,149 size 319x276; Picture "283863143_751404212536178_4947535140145413484_n"
*)